// Mitsubishi GX Works2 project: Class6_Sign&Motor   PLC: Q03UD

PROGRAM SIGN
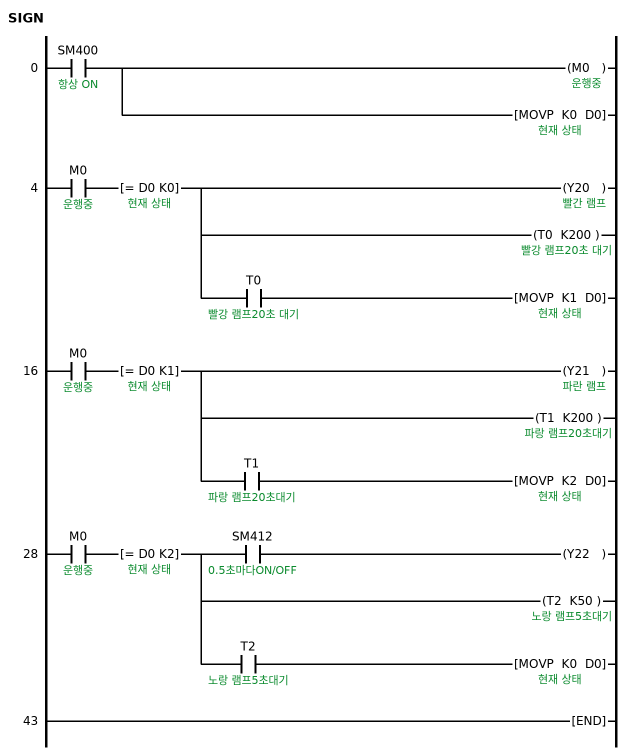
0     LD      SM400  ; 항상 ON
      OUT     M0  ; 운행중
      MOVP    K0 D0  ; 현재 상태
4     LD      M0  ; 운행중
      AND=    D0 K0  ; 현재 상태
      OUT     Y20  ; 빨간 램프
      OUT     T0 K200  ; 빨강 램프20초 대기
      AND     T0  ; 빨강 램프20초 대기
      MOVP    K1 D0
16    LD      M0  ; 운행중
      AND=    D0 K1  ; 현재 상태
      OUT     Y21  ; 파란 램프
      OUT     T1 K200  ; 파랑 램프20초대기
      AND     T1  ; 파랑 램프20초대기
      MOVP    K2 D0
28    LD      M0  ; 운행중
      AND=    D0 K2  ; 현재 상태
      MPS
      AND     SM412  ; 0.5초마다ON/OFF
      OUT     Y22
      MPP
      OUT     T2 K50  ; 노랑 램프5초대기
      AND     T2  ; 노랑 램프5초대기
      MOVP    K0 D0
43    END
END_PROGRAM

PROGRAM MOTOR
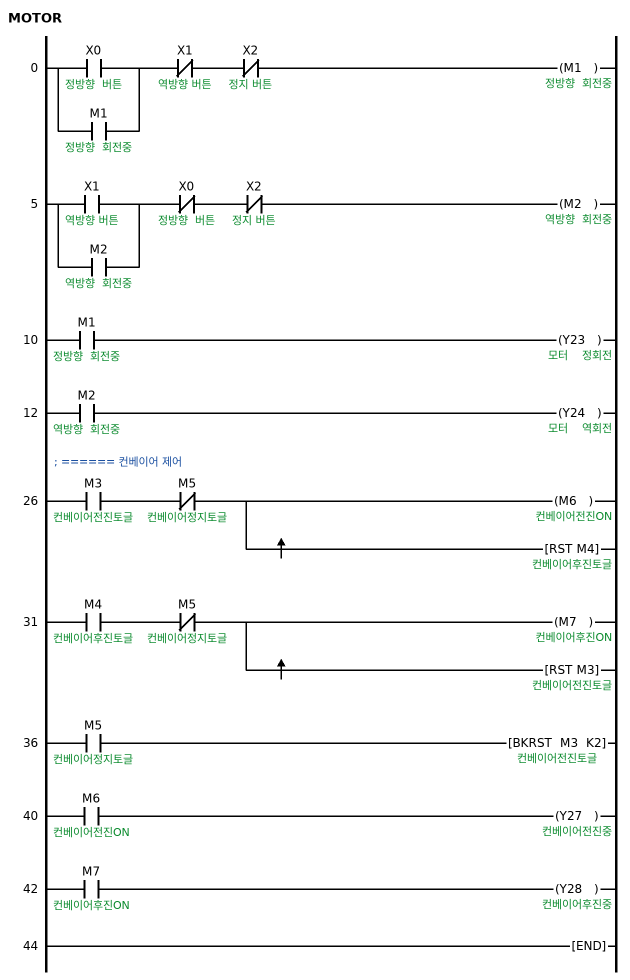
0     LD      X0  ; 정방향  버튼
      OR      M1  ; 정방향  회전중
      ANI     X1  ; 역방향 버튼
      ANI     X2  ; 정지 버튼
      OUT     M1  ; 정방향  회전중
5     LD      X1  ; 역방향 버튼
      OR      M2  ; 역방향  회전중
      ANI     X0  ; 정방향  버튼
      ANI     X2  ; 정지 버튼
      OUT     M2  ; 역방향  회전중
10    LD      M1  ; 정방향  회전중
      OUT     Y23  ; 모터    정회전
12    LD      M2  ; 역방향  회전중
      OUT     Y24  ; 모터    역회전
; ====== 컨베이어 제어
26    LD      M3  ; 컨베이어전진토글
      ANI     M5  ; 컨베이어정지토글
      OUT     M6  ; 컨베이어전진ON
      MEP
      RST     M4  ; 컨베이어후진토글
31    LD      M4  ; 컨베이어후진토글
      ANI     M5  ; 컨베이어정지토글
      OUT     M7  ; 컨베이어후진ON
      MEP
      RST     M3  ; 컨베이어전진토글
36    LD      M5  ; 컨베이어정지토글
      BKRST   M3 K2
40    LD      M6  ; 컨베이어전진ON
      OUT     Y27  ; 컨베이어전진중
42    LD      M7  ; 컨베이어후진ON
      OUT     Y28  ; 컨베이어후진중
44    END
END_PROGRAM

PROGRAM PISTON
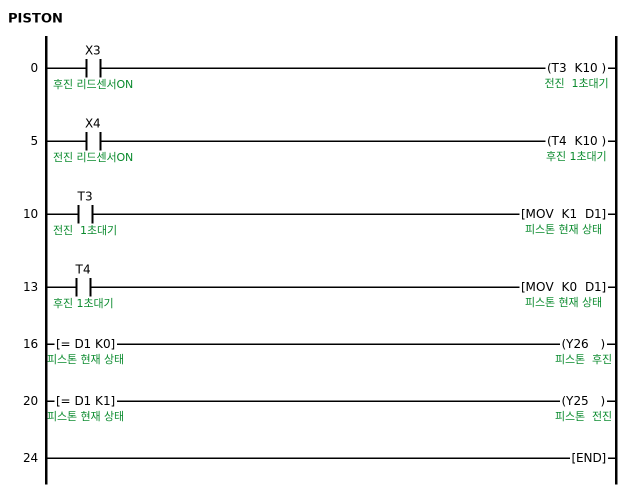
0     LD      X3  ; 후진 리드센서ON
      OUT     T3 K10  ; 전진  1초대기
5     LD      X4  ; 전진 리드센서ON
      OUT     T4 K10  ; 후진 1초대기
10    LD      T3  ; 전진  1초대기
      MOV     K1 D1  ; 피스톤 현재 상태
13    LD      T4  ; 후진 1초대기
      MOV     K0 D1
16    LD=     D1 K0  ; 피스톤 현재 상태
      OUT     Y26  ; 피스톤  후진
20    LD=     D1 K1  ; 피스톤 현재 상태
      OUT     Y25  ; 피스톤  전진
24    END
END_PROGRAM

// device comments not shown above
C0  ; 20회 반복
